FUNCTION_BLOCK CV_FIND_BY_YOLO (* Basic FB with empty ECC *)
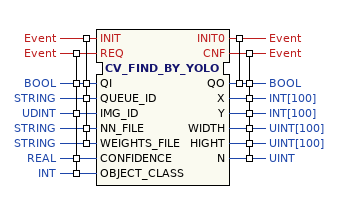
  EVENT_INPUT
    INIT WITH QI, QUEUE_ID, WEIGHTS_FILE, NN_FILE;
    REQ WITH QI, IMG_ID, CONFIDENCE, OBJECT_CLASS;
  END_EVENT
  EVENT_OUTPUT
    INIT0 WITH QO;
    CNF WITH QO, X, Y, WIDTH, HIGHT, N;
  END_EVENT
  VAR_INPUT
    QI : BOOL;
    QUEUE_ID : STRING;
    IMG_ID : UDINT;
    NN_FILE : STRING;
    WEIGHTS_FILE : STRING;
    CONFIDENCE : REAL;
    OBJECT_CLASS : INT;
  END_VAR
  VAR_OUTPUT
    QO : BOOL;
    X : ARRAY [0..99] OF INT;
    Y : ARRAY [0..99] OF INT;
    WIDTH : ARRAY [0..99] OF UINT;
    HIGHT : ARRAY [0..99] OF UINT;
    N : UINT;
  END_VAR
END_FUNCTION_BLOCK
